{attribute 'GeneratedUsingTerminal: EP6601-0002-0018'}
{attribute addProperty BoxType "EP6601-0002-0018"}
{attribute addProperty Id "InfoDataAT %I*InfoData_94A18F5E2"}
{attribute addProperty CRC "2009557638"}
{attribute addProperty Size "2"}
TYPE EP6601_77C76A86 EXTENDS EtcSlaveTerminalBase_947E5A46 :
STRUCT
	{attribute addProperty Name "InfoData"}
	InfoData : InfoData_94A18F5E;
END_STRUCT
END_TYPE

(* stored: Version 1.2.0.0, ProductVersion 3.1.4024.9
   DUT EP6601_77C76A86: Id {6566d8a9-466b-411c-b724-4923b9766621} *)
